ABB RobotStudio station: CakeServer.rspag

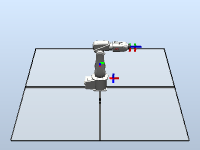
--- station ---
Station Solution2 (saved by RobotStudio 7.0.8460.151)
Controller Vinnie
  mechanical unit ROB_1: IRB120_3_58__01, 6 joints, base frame (0, 0, 0) mm
Layout (positions relative to the parent item):
  - IRB120_3_58__01 [mechanism, from Robots\IRB120_3_58_G_01.rslib] at (0, 0, 0) mm; joint values [0, 0, 0, 0, 0, 0] (rad or m)
Targets, tools, work objects and paths stored in the station and not in the controller backup, written as RAPID:
! task T_ROB1
MODULE MTRN4230_IO_Sample
  PROC MainIO()
    TurnVacOn;
    WaitTime 2;
    TurnVacOff;
    TurnConOnSafely;
    WaitTime 2;
    TurnConOff;
  ENDPROC
  PROC TurnVacOff()
    SetDO DO10_1,0;
  ENDPROC
  PROC TurnConOff()
    SetDO DO10_3,0;
  ENDPROC
  PROC TurnVacOn()
    SetDO DO10_1,1;
  ENDPROC
  PROC TurnConOnSafely()
    SetDO DO10_3,1;
    SetDO DO10_3,0;
  ENDPROC
ENDMODULE


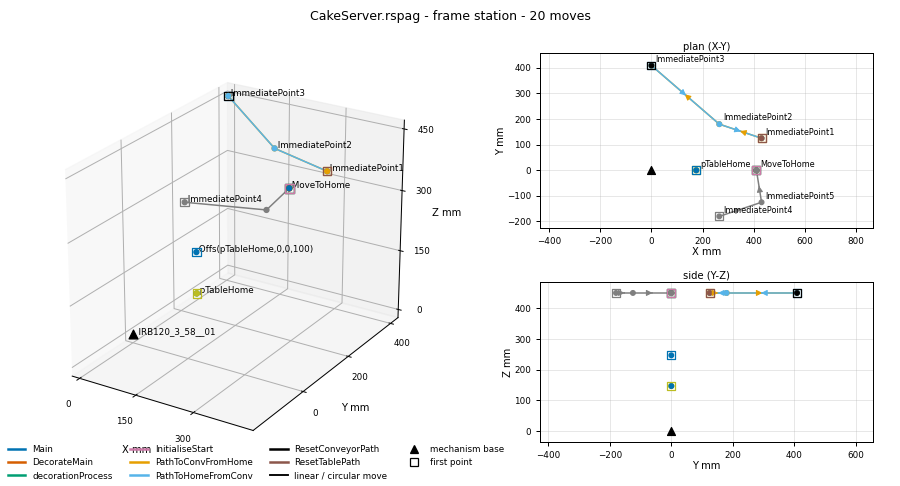
[picture p0: tool path of CakeServer.rspag in frame station, 20 of 38 moves have a stored position in this frame; points joined in program order, loops and branches not executed]
--- Backups/Vinnie/RAPID/TASK1/PROGMOD/CakeShopRobotMain.mod ---
MODULE CakeShopRobotMain
    !***********************************************************
    !
    ! Module: Main robot controller
    ! Author: Rachel Feng, z5112668
    !
    ! Description:
    !   This module is the main controller of all robot movements.
    !   Contains ongoing error checking.
    !   Calls functions to decorate the cake with blocks & icing.
    !   After each pick and place, communicate back to server to see
    !   if decoration is completed.
    !
    !***********************************************************

    ! Interrupts for emergency stops
!    VAR intnum lightCurtain;
!    VAR intnum emergencyStop;
!    VAR intnum emergencyStopMotor;
    VAR num tempConv;
    VAR num response;

    ! Flags to send error message back to GUI
    PERS bool lightCurtainError:=FALSE;
    PERS bool emergencyStopError:=FALSE;
    PERS bool conveyorError:=FALSE;
    PERS bool vacuumError:=FALSE;
    PERS bool clearMessage:=FALSE;

    ! Data received from server
    PERS num letterArrayCopy{3,100,1000};
    PERS num blockArrayCopy{50,7};
    PERS num leftOverArrayCopy{50,6};

    PERS num numLettersCopy;
    PERS num numCoordinatesCopy{100};
    VAR num z_coord:=147.5;

    PERS num numBlocksCopy;
    PERS num numLeftOverCopy;

    ! Flags to check
    PERS bool chocBlocks;
    PERS bool isDecorDone;
    PERS bool letters;
    PERS bool robotMoving;
    PERS bool pauseResume;
    PERS bool stopFlag;

    VAR bool firstConvMove:=FALSE;

    CONST jointtarget removeSingularities := [[0,0,0,0,3,3],[9E+09,9E+09,9E+09,9E+09,9E+09,9E+09]];

    PROC Main()
        ! set up interrups
!        CONNECT timerInt WITH checkTime;
!        ITimer 5,timerInt;
!        ISleep timerInt;

!        CONNECT lightCurtain WITH lTrap;
!        CONNECT emergencyStop WITH eTrap;
!        CONNECT emergencyStopMotor WITH eTrapMotor;

!        ISignalDO\Single,DO_LIGHT_CURTAIN,0,lightCurtain;
!        ISignalDO\Single,DO_ESTOP,1,emergencyStop;
!        ISignalDO\Single,DO_ESTOP2,0,emergencyStopMotor;

        ! Testing stuff
!        ConveyorTestMove01;
!        WaitTime 2;
!        ConveyorTestMove02;
!        WaitTime 2;
!        testVacuumOnOff;
!        WaitTime 2;
!        testSuctionCup;
!        WaitTime 2;
!        DecorTest;
!        WaitTime 2;
!        InkPrintingMain;

        ! stop all functions, return robot arm to home position
        IF stopFlag=TRUE THEN
            turnOffConveyor;
            turnOffGripper;
            turnOffVacuum;
            MoveL MoveToHome,v1000,z100,tool0\WObj:=wobj0;
            StopMove;
            EXIT;
        ENDIF

        ! pause/resume loop
        IF pauseResume=FALSE THEN
            StopMove;
            IF DOutput(DO10_3)=1 THEN
                turnOffConveyor;
                tempConv:=1;
            ENDIF
            WHILE pauseResume=FALSE DO
                ! do nothing
            ENDWHILE
            IF tempConv=1 THEN
                turnOnConveyor;
                tempConv:=0;
            ENDIF
            StartMove;
        ENDIF

        ! move conveyor for first choc block picture
        IF firstConvMove=FALSE THEN
            setDirToRobot;
            turnOnConveyor;
            WaitTime 5;
            turnOffConveyor;
            firstConvMove:=TRUE;
            robotMoving:=FALSE;
        ENDIF

        ! main decoration routine
        IF chocBlocks=TRUE THEN
            DecorateMain blockArrayCopy;
            DecorateMain leftOverArrayCopy;
            chocBlocks:=FALSE;
            turnOnConveyor;
            WaitTime 1;
            turnOffConveyor;
            robotMoving:=FALSE;
        ENDIF

        ! main lettering/icing routine
        IF letters=TRUE THEN
            draw_letter letterArrayCopy, sizes ,167;
            letters:=FALSE;
        ENDIF

        ! delete interrupts (temp)
!        IDelete timerInt;
!        IDelete emergencyStop;
!        IDelete emergencyStopMotor;
!        IDelete lightCurtain;
    ENDPROC

!    ! light curtain trap routine
!    TRAP lTrap
!        ! stop the robot & conveyor
!        StopMove;
!        IF DOutput(DO10_3)=1 THEN
!            turnOffConveyor;
!            tempConv:=1;
!        ENDIF
!        ! print message to gui
!        lightCurtainError:=TRUE;
!        ! print message to flex pendant
!        TPErase;
!        TPWrite "Light curtain obstruction";
!        TPReadFK response,"Please remove obstruction",stEmpty,stEmpty,stEmpty,"No","Fixed";
!        IF response=4 THEN
!            TPErase;
!            TPWrite "Exiting program...";
!            WaitTime 2;
!            EXIT;
!        ELSEIF response=5 THEN
!            TPErase;
!            TPWrite "Resuming...";
!            clearMessage:=TRUE;
!        ENDIF
!        StartMove;
!        IF tempConv=1 THEN
!            turnOnConveyor;
!            tempConv:=0;
!        ENDIF
!        lightCurtainError:=FALSE;
!        RETURN ;
!    ENDTRAP

!    ! emergency stop interrupt for red buttons except motor
!    TRAP eTrap
!        ! stop the robot
!        StopMove;
!        IF DOutput(DO10_3)=1 THEN
!            turnOffConveyor;
!            tempConv:=1;
!        ENDIF
!        ! print message to gui
!        emergencyStopError:=TRUE;
!        ! print message to flex pendant
!        TPErase;
!        TPWrite "Emergency stop!";
!        TPWrite "Please remove any obstructions and hazards from the robot.";
!        TPWrite "Don't forget to reset the light curtain.";
!        TPReadFK response,"Restart?",stEmpty,stEmpty,stEmpty,"No","Yes";
!        IF response=4 THEN
!            TPErase;
!            TPWrite "Exiting program...";
!            WaitTime 2;
!            EXIT;
!        ELSEIF response=5 THEN
!            TPErase;
!            TPWrite "Resuming...";
!            clearMessage:=TRUE;
!        ENDIF
!        StartMove;
!        IF tempConv=1 THEN
!            turnOnConveyor;
!            tempConv:=0;
!        ENDIF
!        emergencyStopError:=FALSE;
!        RETURN ;
!    ENDTRAP

!    ! emergency stop interrupt for motor button
!    TRAP eTrapMotor
!        ! stop the robot
!        StopMove;
!        IF DOutput(DO10_3)=1 THEN
!            turnOffConveyor;
!            tempConv:=1;
!        ENDIF
!        ! print message to gui
!        emergencyStopError:=TRUE;
!        ! print message to flex pendant
!        TPErase;
!        TPWrite "Motor stop!";
!        TPWrite "Please remove any obstructions and hazards from the robot.";
!        TPWrite "Don't forget to reset the light curtain.";
!        TPReadFK response,"Restart?",stEmpty,stEmpty,stEmpty,"No","Yes";
!        IF response=4 THEN
!            TPErase;
!            TPWrite "Exiting program...";
!            WaitTime 2;
!            EXIT;
!        ELSEIF response=5 THEN
!            TPErase;
!            TPWrite "Resuming...";
!            clearMessage:=TRUE;
!        ENDIF
!        StartMove;
!        IF tempConv=1 THEN
!            turnOnConveyor;
!            tempConv:=0;
!        ENDIF
!        emergencyStopError:=FALSE;
!        RETURN ;
!    ENDTRAP

ENDMODULE

--- Backups/Vinnie/RAPID/TASK1/PROGMOD/ConveyorController.mod ---
MODULE ConveyorController
    !***********************************************************
    !
    ! Module: Conveyor Controller
    ! Author: Rachel Feng, z5112668
    !
    ! Description:
    !   This is a module containing all conveyor commands to be called by other modules
    !
    !***********************************************************

    ! Response from error provided from the user
    !VAR num convResp;
    ! Error number for conveyor movement fail
    !VAR errnum CONV_MOVE_ERR:=-1;

    PROC turnOnConveyor()
        !BookErrNo CONV_MOVE_ERR;
        ! if conveyor status (constat) is 1, good to go
        !IF DI10_1=1 THEN
            SetDO DO10_3,1;
        !ELSE
        !    turnOffConveyor;
        !    RAISE CONV_MOVE_ERR;
        !ENDIF

!    ERROR
!        ! Conveyor error: occurs when attempt to turn on conveyor occured when IO/Light Curtain/Cage is not ready/set up
!        IF ERRNO=CONV_MOVE_ERR THEN
!            ! print to gui
!            conveyorError:=TRUE;
!            ! print message to flex pendant
!            TPErase;
!            TPWrite "Please check light curtain and conveyor guard then restart conveyor";
!            TPReadFK convResp,"Checked?",stEmpty,stEmpty,stEmpty,"No","Yes";
!            IF convResp=4 THEN
!                convResp:=0;
!                TPErase;
!                TPWrite "Exiting...";
!                EXIT;
!            ELSEIF convResp=5 THEN
!                convResp:=0;
!                clearMessage:=TRUE;
!                TPErase;
!                TPWrite "Retrying...";
!                conveyorError:=FALSE;
!                RETRY;
!            ENDIF
!        ENDIF
    ENDPROC

    PROC turnOffConveyor()
        SetDO DO10_3,0;
    ENDPROC

    PROC setDirToRobot()
        SetDO DO10_4,1;
    ENDPROC

    PROC setDirFromRobot()
        ! default
        SetDO DO10_4,0;
    ENDPROC
ENDMODULE

--- Backups/Vinnie/RAPID/TASK1/PROGMOD/DecorationPickAndPlace.mod ---
MODULE DecorationPickAndPlace
    !***********************************************************
    !
    ! Module: Decoration Movement Code for Robot
    ! Author: Dylan Dam, z5115759
    !
    ! Description:
    !    This module is responsible for the pick and place for the qwirkle decoration.
    !    The function takes an array that contains the start and end coordinates of the
    !    blocks as well as it's orientation. The robot then moves via a set path that is
    !    defined and proceeds to move to the location of the block on the conveyor belt.
    !    After picking up the block the arm traverses back via the same path and places
    !    the block down. There is a function that rotates axis 6 for blocks that are
    !    orientated differently. After the execution of the place and drop the robot
    !    moves back to the home position.
    !
    ! Inputs:
    !   array - a nx6 or nx7 matrix data, recevied from GUI part, see GUI for more info
    !
    !***********************************************************

    ! Custom waypoints that I have selected
    CONST robtarget ImmediatePoint1:=[[430,125,450],[0,0,1,0],[0,-1,0,0],[9E+09,9E+09,9E+09,9E+09,9E+09,9E+09]];
    CONST robtarget ImmediatePoint2:=[[265,180,450],[0,0,1,0],[0,-1,0,0],[9E+09,9E+09,9E+09,9E+09,9E+09,9E+09]];
    CONST robtarget ImmediatePoint3:=[[0,409,450],[0,0,1,0],[1,-1,1,0],[9E+09,9E+09,9E+09,9E+09,9E+09,9E+09]];
    CONST robtarget ImmediatePoint4:=[[265,-180,450],[0,0,1,0],[1,-1,1,0],[9E+09,9E+09,9E+09,9E+09,9E+09,9E+09]];
    CONST robtarget ImmediatePoint5:=[[430,-125,450],[0,0,1,0],[1,-1,1,0],[9E+09,9E+09,9E+09,9E+09,9E+09,9E+09]];
    CONST robtarget MoveToHome:=[[410,0,450],[0,0,-1,0],[0,0,-1,0],[9E+09,9E+09,9E+09,9E+09,9E+09,9E+09]];
    ! Offset for the end-effector
    CONST num offSet := 75;
    !Dummy Array for Testing
    !CONST num qwirkleArray{4,7} := [[175,0,147,0,409,22.1,45],[548.6,0,147,0,409,22.1,0],[175,520,147,0,409,22.1,-45],[175,-300,147,0,409,22.1,-45]];
    CONST num qwirkleArray{1,7} := [[175,-50,147,0,409,22.1,-89]];

    PROC DecorateMain(num array{*,*})
        TPWRite "Decorating...";
        MoveAbsJ removeSingularities,v400,fine,tool0;
        MoveL MoveToHome,v1000,z100,tool0\WObj:=wobj0;
        WaitTime 1;
        decorationProcess array;
        WaitTime 1;
        MoveL MoveToHome,v1000,z100,tool0\WObj:=wobj0;
        WaitTime 1;
    ENDPROC

    PROC decorationProcess(num array{*,*})

        VAR num xStart;
        VAR num yStart;
        VAR num zStart;
        VAR num xEnd;
        VAR num yEnd;
        VAR num zEnd;
        VAR num orientation;
        VAR robtarget qwirkleLocation;
        VAR robtarget qwirklePlacement;

        FOR a FROM 1 TO Dim(array,1) DO
            ! This part reads in the first line.
            xStart := array{a,4};
            yStart := array{a,5};
            IF xStart = 0 AND yStart = 0 THEN
                ExitCycle;
            ENDIF
            !zStart := array{a,6}+offSet;
            zStart := 22.1+offSet;
            xEnd := array{a,1};
            yEnd := array{a,2};
            zEnd := 147+offSet;
            orientation := array{a,7};

            qwirkleLocation := [[xStart,yStart,zStart],[0,0,1,0],[0,0,0,0],[9E+09,9E+09,9E+09,9E+09,9E+09,9E+09]];
            qwirklePlacement :=[[xEnd,yEnd,zEnd],[0,0,1,0],[0,0,0,0],[9E+09,9E+09,9E+09,9E+09,9E+09,9E+09]];

            PathToConvFromHome;
            MoveL qwirkleLocation,v1000,z100,tool0\WObj:=wobj0;
            WaitTime 1;
            turnOnVacuum;
            turnOnGripper;
            ResetConveyorPath;
            PathToHomeFromConv;
            WaitTime 1;
            MoveL qwirklePlacement,v1000,z100,tool0\WObj:=wobj0;
            RotateTool orientation,qwirklePlacement;
            IF (yEnd < -400) THEN
                LeftSidePath;
            ELSE
                MoveL MoveToHome,v1000,z100,tool0\WObj:=wobj0;
            ENDIF

        ENDFOR

    ENDPROC

    PROC InitialiseStart()
        MoveL MoveToHome,v1000,z100,tool0\WObj:=wobj0;
    ENDPROC

    PROC PathToConvFromHome()
            MoveL ImmediatePoint1,v1000,z100,tool0\WObj:=wobj0;
            MoveL ImmediatePoint2,v1000,z100,tool0\WObj:=wobj0;
            MoveL ImmediatePoint3,v1000,z100,tool0\WObj:=wobj0;
    ENDPROC

    PROC PathToHomeFromConv()
        MoveL ImmediatePoint3,v1000,z100,tool0\WObj:=wobj0;
        MoveL ImmediatePoint2,v1000,z100,tool0\WObj:=wobj0;
        MoveL ImmediatePoint1,v1000,z100,tool0\WObj:=wobj0;
    ENDPROC
    PROC ResetConveyorPath()
        MoveL ImmediatePoint3,v1000,z100,tool0\WObj:=wobj0;
    ENDPROC
    PROC ResetTablePath()
        MoveL ImmediatePoint1,v1000,z100,tool0\WObj:=wobj0;
    ENDPROC

    PROC RotateTool(num Orientation,robtarget a)
        IF Orientation > 90 THEN
            Orientation := 90 - Orientation;
            MoveL RelTool(a,0,0,0,\Rz:= Orientation),v1000,fine,tool0\WObj:=wobj0;
            WaitTime 1;
            turnOffGripper;
            turnOffVacuum;
            WaitTime 1;
        ELSE
            MoveL RelTool(a,0,0,0,\Rz:= Orientation),v1000,fine,tool0\WObj:=wobj0;
            WaitTime 1;
            turnOffGripper;
            turnOffVacuum;
            WaitTime 1;
        ENDIF

    ENDPROC

    PROC LeftSidePath()

        MoveL ImmediatePoint4,v1000,z100,tool0\WObj:=wobj0;
        MoveL ImmediatePoint5,v1000,z100,tool0\WObj:=wobj0;
        MoveL MoveToHome,v1000,z100,tool0\WObj:=wobj0;


    ENDPROC

ENDMODULE

--- Backups/Vinnie/RAPID/TASK1/PROGMOD/InkPrinting.mod ---
MODULE InkPrinting
    !***********************************************************
    !
    ! Module: Ink Printing
    ! Author: Mike Ni, z5083683
    !
    ! Description:
    !   Runs program to move TCP along a given trajectory with a given speed decided by boldness of letter
    !
    ! Input:
    !   data_matrix - a 3xnxm matrix data, recevied from GUI part, see GUI for more info
    !   z_coor - the z coordinate for ink printing, assume to be 147.5
    !
    !***********************************************************

    PERS num x_array{135,1};
    PERS num y_array{135,1};
    PERS num z_array;
    PERS num letterArray{3,8,135};
    PERS num sizes{8};
    ! boldness 0 - unbolded, 1 - bolded
    PERS num bolded{8};
    PERS num boldness;
    ! The Main procedure. When you select 'PP to Main' on the FlexPendant, it will go to this procedure.
    PROC InkPrintingMain()

        ! This is a procedure defined in a System Module, so you will have access to it.
        ! This will move the robot to its calibration.
         MoveToCalibPos;

        ! Call a procedure that we have defined below.
         MoveJSample;

        ! Call another procedure that we have defined.
        ! MoveLSample;
        Path_10;
        !draw_path;
        draw_letter letterArray, sizes, 167;
        !Path_10;

        ! Call another procedure, but provide some input arguments.
        ! VariableSample pTableHome, 100, 100, 0, v100, fine;

        MoveToCalibPos;
    ENDPROC

    PROC draw_path()
        VAR num x;
        VAR num y;
        VAR num z;
        VAR num x_next;
        VAR num y_next;
        VAR pos curr;
        VAR pos next;
        VAR pos prev;
        VAR robtarget pathLoc;
        VAR num distance_from_next;
        VAR num displacement;
        VAR num time_req;
        FOR i FROM 1 TO DIM(x_array,1) DO
            x := x_array{i, 1};
            y := y_array{i, 1};
            ! find next point, except for last point
            IF i <> DIM(x_array, 1) THEN
                x_next := x_array{i+1, 1};
                y_next := y_array{i+1, 1};
            ELSE
                x_next := x;
                y_next := y;
            ENDIF
            z := z_array;
            curr := [x, y, z];
            next := [x_next, y_next, z];
            distance_from_next := Distance(curr, next);
            ! find previous point, start from i = 2
            IF i > 1 THEN
                prev := [x_array{i-1, 1}, x_array{i-1, 1}, z];
                displacement :=  Distance(CPos(\Tool:=tSCup \WObj:=wobj0), curr);
            ENDIF
            pathLoc := [[x, y, z],[0,0,-1,0],[0,0,0,0],[9E9,9E9,9E9,9E9,9E9,9E9]];
            ! check boldness to set speed. 0 - 50mm/s; 1 - 100mm/s
            IF boldness = 0 THEN
                time_req := displacement / 50;
                MoveL pathLoc, v50, z0, tSCup;
                !MoveL pathLoc, v50, \T:=1, fine, tSCup;
            ELSE
                time_req := displacement / 100;
                MoveL pathLoc, v100, z0, tSCup;
                !MoveL pathLoc, v100, \T:= 1, fine, tSCup;
            ENDIF
            !if next point is very far away, move tcp away from object surface
            IF distance_from_next > 15 THEN
                pathLoc := [[x, y, z+50],[0,0,-1,0],[0,0,0,0],[9E9,9E9,9E9,9E9,9E9,9E9]];
                MoveL pathLoc, vmax, \T:=0.1, fine, tSCup;
            ENDIF
        ENDFOR
        !move tcp away once all movement done
        pathLoc := [[x, y, z+10],[0,0,-1,0],[0,0,0,0],[9E9,9E9,9E9,9E9,9E9,9E9]];
        MoveL pathLoc, vmax, \T:=0.1, fine, tSCup;
    ENDPROC

    !use "draw_letter data_matrix" to run
    PROC draw_letter(num data_matrix{*,*,*}, num sizeOfLetter{*}, num z_coor)
        VAR num x;
        VAR num y;
        VAR num z;
        VAR num x_next;
        VAR num y_next;
        VAR pos curr;
        VAR pos next;
        VAR pos prev;
        VAR robtarget pathLoc;
        VAR num distance_from_next;
        VAR num displacement;
        VAR num time_req;
        VAR num bolded;
        VAR speeddata speed;
        MoveAbsJ removeSingularities,v400,fine,tool0;
        FOR index FROM 1 TO DIM(data_matrix,2) DO
            bolded := data_matrix{1,index,1};
            IF bolded = 0 THEN
                speed := [50, 500, 5000, 1000];
            ELSE
                speed := [100, 500, 5000, 1000];
            ENDIF
            FOR i FROM 1 TO sizeOfLetter{index} DO
                x := data_matrix{2,index,i};
                y := data_matrix{3,index,i};

                ! find next point, except for last point
                IF i <> DIM(data_matrix,3) THEN
                    x_next := data_matrix{2,index,i+1};
                    y_next := data_matrix{3,index,i+1};
                ELSE
                    x_next := x;
                    y_next := y;
                ENDIF
                z := z_coor;
                curr := [x, y, z];
                next := [x_next, y_next, z];
                distance_from_next := Distance(curr, next);
                ! find previous point, start from i = 2
                IF i > 1 THEN
                    prev := [data_matrix{2,index,i-1}, data_matrix{3,index,i-1}, z];
                    displacement :=  Distance(CPos(\Tool:=tSCup \WObj:=wobj0), curr);
                ENDIF
                pathLoc := [[x, y, z],[0,0,-1,0],[0,0,0,0],[9E9,9E9,9E9,9E9,9E9,9E9]];
                ! check boldness to set speed. 0 - 50mm/s; 1 - 100mm/s

                MoveL pathLoc, speed, z0, tSCup;

                !if next point is very far away, move tcp away from object surface
                IF distance_from_next > 15 THEN
                    pathLoc := [[x, y, z+50],[0,0,-1,0],[0,0,0,0],[9E9,9E9,9E9,9E9,9E9,9E9]];
                    MoveL pathLoc, vmax, \T:=0.1, fine, tSCup;
                ENDIF
            ENDFOR
            !move tcp away once all movement done
            pathLoc := [[x, y, z+10],[0,0,-1,0],[0,0,0,0],[9E9,9E9,9E9,9E9,9E9,9E9]];
            MoveL pathLoc, vmax, \T:=0.1, fine, tSCup;
        ENDFOR
    ENDPROC

    PROC Path_10()
        !Defines the trajectory coordinates
        VAR num step_count := 0;
        bolded := [0,1,0,1,0,1,0,1];
        boldness := 0;
        x_array := [
        [347.3852228],
        [340.1824253],
        [332.9796278],
        [325.7768303],
        [319.2288325],
        [312.026035],
        [304.8232375],
        [309.4068359],
        [315.9548336],
        [322.5028314],
        [329.0508291],
        [335.5988269],
        [342.1468246],
        [300.2396391],
        [306.7876368],
        [313.9904343],
        [321.1932318],
        [327.7412296],
        [334.9440271],
        [341.4920249],
        [302.8588381],
        [308.7520361],
        [315.3000339],
        [321.8480316],
        [328.3960294],
        [334.9440271],
        [341.4920249],
        [304.1684377],
        [304.8232375],
        [304.8232375],
        [304.8232375],
        [350.0044219],
        [344.111224],
        [336.9084264],
        [329.7056289],
        [322.5028314],
        [315.3000339],
        [308.0972363],
        [348.0400226],
        [340.8372251],
        [333.6344276],
        [326.43163],
        [325.1220305],
        [325.7768303],
        [331.0152285],
        [337.5632262],
        [344.7660237],
        [324.4672307],
        [319.2288325],
        [312.6808348],
        [306.132837],
        [302.8588381],
        [302.2040384],
        [305.4780372],
        [312.6808348],
        [319.8836323],
        [302.2040384],
        [307.4424366],
        [312.6808348],
        [319.2288325],
        [325.7768303],
        [332.324828],
        [338.8728258],
        [344.7660237],
        [304.8232375],
        [311.3712352],
        [318.5740327],
        [325.7768303],
        [332.324828],
        [338.8728258],
        [350.0044219],
        [343.4564242],
        [336.2536267],
        [329.0508291],
        [321.8480316],
        [314.6452341],
        [350.0044219],
        [336.9084264],
        [341.4920249],
        [348.6948224],
        [304.1684377],
        [310.7164354],
        [317.919233],
        [325.1220305],
        [332.324828],
        [336.2536267],
        [336.2536267],
        [329.7056289],
        [323.1576312],
        [316.6096334],
        [310.7164354],
        [304.8232375],
        [351.3140215],
        [346.0756233],
        [348.6948224],
        [348.6948224],
        [312.6808348],
        [307.4424366],
        [306.132837],
        [310.7164354],
        [317.2644332],
        [323.8124309],
        [329.0508291],
        [334.2892273],
        [340.1824253],
        [343.4564242],
        [349.3496222],
        [351.3140215],
        [348.6948224],
        [342.8016244],
        [335.5988269],
        [329.0508291],
        [322.5028314],
        [315.9548336],
        [309.4068359],
        [304.8232375],
        [305.4780372],
        [310.7164354],
        [325.7768303],
        [321.8480316],
        [315.3000339],
        [308.7520361],
        [306.7876368],
        [310.0616357],
        [316.6096334],
        [323.1576312],
        [330.3604287],
        [336.9084264],
        [343.4564242],
        [348.6948224],
        [349.3496222],
        [344.7660237],
        [338.218026],
        [331.6700282],
        [324.4672307]
        ];

        y_array := [
        [137.4530852],
        [137.4530852],
        [137.4530852],
        [137.4530852],
        [136.800876],
        [136.800876],
        [136.800876],
        [131.5832025],
        [130.2787841],
        [128.9743658],
        [127.6699474],
        [126.3655291],
        [125.0611107],
        [104.842626],
        [106.7992536],
        [106.7992536],
        [106.7992536],
        [106.7992536],
        [106.7992536],
        [107.4514628],
        [108.103672],
        [111.3647179],
        [113.3213454],
        [115.277973],
        [117.2346005],
        [118.5390189],
        [119.8434372],
        [94.40727912],
        [87.23297812],
        [80.05867712],
        [72.88437611],
        [80.7108863],
        [83.97193221],
        [83.97193221],
        [83.97193221],
        [83.97193221],
        [83.97193221],
        [83.97193221],
        [61.14461083],
        [61.14461083],
        [61.14461083],
        [60.49240165],
        [53.97030983],
        [46.79600882],
        [42.23054455],
        [41.57833537],
        [41.57833537],
        [46.79600882],
        [41.57833537],
        [40.92612618],
        [42.88275373],
        [48.75263637],
        [55.27472819],
        [61.14461083],
        [61.14461083],
        [61.14461083],
        [29.1863609],
        [24.62089663],
        [20.05543235],
        [17.44659562],
        [15.48996808],
        [12.88113135],
        [9.620085438],
        [6.359039527],
        [3.750202798],
        [4.40241198],
        [4.40241198],
        [4.40241198],
        [3.750202798],
        [5.706830344],
        [24.62089663],
        [27.22973336],
        [27.22973336],
        [27.22973336],
        [27.22973336],
        [26.57752417],
        [-25.5992104],
        [-30.81688386],
        [-25.5992104],
        [-25.5992104],
        [-26.25141958],
        [-25.5992104],
        [-25.5992104],
        [-25.5992104],
        [-25.5992104],
        [-19.72932776],
        [-12.55502676],
        [-10.59839921],
        [-13.85944512],
        [-17.12049103],
        [-20.38153694],
        [-24.29479204],
        [-36.6867665],
        [-41.90443996],
        [-48.42653178],
        [-55.60083278],
        [-40.60002159],
        [-45.16548587],
        [-51.68757769],
        [-57.55746033],
        [-58.20966951],
        [-56.25304197],
        [-51.68757769],
        [-47.12211341],
        [-43.20885832],
        [-68.64501643],
        [-71.90606234],
        [-78.42815416],
        [-84.95024598],
        [-88.21129189],
        [-88.21129189],
        [-85.60245516],
        [-84.95024598],
        [-87.55908271],
        [-86.90687353],
        [-81.68920007],
        [-74.51489907],
        [-69.94943479],
        [-77.1237358],
        [-100.6032664],
        [-101.9076847],
        [-105.1687306],
        [-111.6908225],
        [-118.2129143],
        [-120.1695418],
        [-120.821751],
        [-120.821751],
        [-120.1695418],
        [-118.8651235],
        [-114.2996592],
        [-107.7775674],
        [-102.5598939],
        [-101.2554755],
        [-100.6032664],
        [-100.6032664]
        ];

        sizes:=[27,11,18,20,16,13,14,16];
        z_array := 147;
        FOR i FROM 1 TO 27 DO
            letterArray{1,1,1} := bolded{1};
            letterArray{2,1,i} := x_array{i+step_count,1};
            letterArray{3,1,i} := y_array{i+step_count,1};
        ENDFOR
        step_count := 27;
        FOR i FROM 1 TO 11 DO
            letterArray{1,2,1} := bolded{2};
            letterArray{2,2,i} := x_array{i+step_count,1};
            letterArray{3,2,i} := y_array{i+step_count,1};
        ENDFOR
        step_count := 38;
        FOR i FROM 1 TO 18 DO
            letterArray{1,3,1} := bolded{3};
            letterArray{2,3,i} := x_array{i+step_count,1};
            letterArray{3,3,i} := y_array{i+step_count,1};
        ENDFOR
        step_count := 56;
        FOR i FROM 1 TO 20 DO
            letterArray{1,4,1} := bolded{4};
            letterArray{2,4,i} := x_array{i+step_count,1};
            letterArray{3,4,i} := y_array{i+step_count,1};
        ENDFOR
        step_count := 76;
        FOR i FROM 1 TO 16 DO
            letterArray{1,5,1} := bolded{5};
            letterArray{2,5,i} := x_array{i+step_count,1};
            letterArray{3,6,i} := y_array{i+step_count,1};
        ENDFOR
        step_count := 92;
        FOR i FROM 1 TO 13 DO
            letterArray{1,6,1} := bolded{6};
            letterArray{2,6,i} := x_array{i+step_count,1};
            letterArray{3,6,i} := y_array{i+step_count,1};
        ENDFOR
        step_count := 105;
        FOR i FROM 1 TO 14 DO
            letterArray{1,7,1} := bolded{7};
            letterArray{2,7,i} := x_array{i+step_count,1};
            letterArray{3,7,i} := y_array{i+step_count,1};
        ENDFOR
        step_count := 119;
        FOR i FROM 1 TO 16 DO
            letterArray{1,8,1} := bolded{8};
            letterArray{2,8,i} := x_array{i+step_count,1};
            letterArray{3,8,i} := y_array{i+step_count,1};
        ENDFOR
        !FOR i FROM 1 TO DIM(x_array, 1) DO
        !    letterArray{2,1,i} := x_array{i,1};
        !    letterArray{3,1,i} := y_array{i,1};
        !ENDFOR
    ENDPROC

    PROC MoveJSample()

        ! 'MoveJ' executes a joint motion towards a robtarget. This is used to move the robot quickly from one point to another when that
        !   movement does not need to be in a straight line.
        ! 'pTableHome' is a robtarget defined in system module. The exact location of this on the table has been provided to you.
        ! 'v100' is a speeddata variable, and defines how fast the robot should move. The numbers is the speed in mm/sec, in this case 100mm/sec.
        ! 'fine' is a zonedata variable, and defines how close the robot should move to a point before executing its next command.
        !   'fine' means very close, other values such as 'z10' or 'z50', will move within 10mm and 50mm respectively before executing the next command.
        ! 'tSCup' is a tooldata variable. This has been defined in a system module, and represents the tip of the suction cup, telling the robot that we
        !   want to move this point to the specified robtarget. Please be careful about what tool you use, as using the incorrect tool will result in
        !   the robot not moving where you would expect it to. Generally you should be using
        MoveJ pTableHome, v100, \T:=0.5, fine, tSCup;

    ENDPROC

    PROC MoveLSample()

        ! 'MoveL' will move in a straight line between 2 points. This should be used as you approach to pick up a chocolate
        ! 'Offs' is a function that is used to offset an existing robtarget by a specified x, y, and z. Here it will be offset 100mm in the positive z direction.
        !   Note that function are called using brackets, whilst procedures and called without brackets.
        MoveL Offs(pTableHome, 0, 0, 100), v100, fine, tSCup;

    ENDPROC

    PROC VariableSample(robtarget target, num x_offset, num y_offset, num z_offset, speeddata speed, zonedata zone)

        ! Call 'MoveL' with the input arguments provided.
        MoveL Offs(target, x_offset, y_offset, z_offset), speed, zone, tSCup;

    ENDPROC

ENDMODULE

--- Backups/Vinnie/RAPID/TASK1/PROGMOD/VacuumController.mod ---
MODULE VacuumController
    !***********************************************************
    !
    ! Module: Vacuum Controller
    ! Author: Rachel Feng, z5112668
    !
    ! Description:
    !   This is a module containing all vacuum commands to be called by other modules
    !
    !***********************************************************

    ! Response from error provided by the user
    VAR num vacResp;
    ! Error number for suction cup fail
    VAR errnum SUCTION_CUP_ERR:=-1;
    ! Timer interrupt
!    VAR intnum timerInt;

    PROC turnOnVacuum()
        SetDO DO10_1,1;
        !        IWatch timerInt;
    ENDPROC

    PROC turnOffVacuum()
!        ISleep timerInt;
        turnOffGripper;
        SetDO DO10_1,0;
    ENDPROC

    PROC turnOnGripper()
        BookErrNo SUCTION_CUP_ERR;
        IF DOutput(DO10_1)=1 THEN
            SetDO DO10_2,1;
        ELSE
            RAISE SUCTION_CUP_ERR;
        ENDIF

    ERROR
        ! Suction cup error: occurs when attempt to activate suction cup occured before vacuum pump activation
        IF ERRNO=SUCTION_CUP_ERR THEN
            ! print message to gui
            vacuumError:=TRUE;
            ! print message to flex pendant
            TPErase;
            TPReadFK vacResp,"Do you want to turn on vacuum?",stEmpty,stEmpty,stEmpty,"No","Yes";
            IF vacResp=4 THEN
                vacResp:=0;
                TPErase;
                TPWrite "Exiting...";
                EXIT;
            ELSEIF vacResp=5 THEN
                vacResp:=0;
                clearMessage:=TRUE;
                TPErase;
                TPWrite "Turning on vacuum";
                turnOnVacuum;
                vacuumError:=FALSE;
                RETRY;
            ENDIF
        ENDIF


    ENDPROC

    PROC turnOffGripper()
        SetDO DO10_2,0;
    ENDPROC

!    TRAP checkTime
!        TPErase;
!        TPWrite "Vacuum was on for too long...";
!        TPWrite "Turning off...";
!        turnOffVacuum;
!        RETURN ;
!    ENDTRAP
ENDMODULE

--- Backups/Vinnie/RAPID/TASK1/SYSMOD/MTRN_Rob_Data.sys ---
MODULE MTRN_Rob_Data (SYSMODULE, NOSTEPIN, READONLY)

 ! PREDEFINED DATA AND ROBOT CELL INFORMATION
 !*******************************************

 ! For the ABB IRB120 Robot in the Mechatronics Blockhouse Lab for the MTRN4230 Robotics Course 2014

 ! TARGETS
 !********

 ! Calibrate Position for all Joints
 CONST jointtarget jtCalibPos:=[[0,0,0,0,0,0],[9E+09,9E+09,9E+09,9E+09,9E+09,9E+09]];

  ! Home Position
 CONST jointtarget jtHomePos:=[[-90,0,0,0,0,0],[9E+09,9E+09,9E+09,9E+09,9E+09,9E+09]];

 ! Home Position of the Table (T1) with tSCup touching Table
 CONST robtarget pTableHome:=[[175,0,147],[0,0,-1,0],[0,0,0,0],[9E+09,9E+09,9E+09,9E+09,9E+09,9E+09]];

 ! Home Position of the Conveyor (C1) with tSCup touching Conveyor
 CONST robtarget pConvHome:=[[0,409,22],[0,-0.7071068,0.7071068,0],[0,0,0,0],[9E+09,9E+09,9E+09,9E+09,9E+09,9E+09]];

 ! Table & Conveyor Dimensions, References & Extent limits as Follows (X,Y,Z in mm):
 !
 !                                                       Conveyor Frame
 !       ------>Y                                   |<-------- 616 -------->|
 !       |                                          |   | Conveyor Belt |   |
 !       |                                          |   |<---- 450 ---->|   |
 !       |                            ||    --------|   |               |   |
 !       v                            \/    |------||   |   0,409,22    |   |
 !       X             Robot Centre  ---->  ||  + |||   |      +        |   |
 !                                          ||    |||   |      C1       |   |
 !     Robot Centre to edge of Table=129    -|    |_|   |               |   |
 !   ----------------------------------------|    |-----------------------------------
 !   |                                /\      ----                                   |
 !   |                                ||      |  |                                   |
 !   |     175,-520,147                     175,0,147                  175,520,147   |
 !   |           +                              +                           +        |
 !   |           T2                             T1                          T3       |
 !   |                                                                               |
 !   |                                                                               |
 !   |                                    548.6,0,147                                |
 !   |                                          +                                    |
 !   |                                          T4                                   |
 !   |                                                                               |
 !   ---------------------------------------------------------------------------------

 ! TOOL DATA
 !**********

 ! Suction Cup Tool Data
 PERS tooldata tSCup:=[TRUE,[[0,0,65],[1,0,0,0]],[0.5,[0,0,20],[1,0,0,0],0,0,0]];
 !
 ! Suction Cup Face is 65mm in Z direction from Tool0

 ! LOAD DATA
 !**********

 ! Chocolate Bar Load Data
 PERS loaddata loChoc:=[0.035,[0,0,3],[1,0,0,0],0,0,0];

 !
 ! Chocolate Bar Weight    : 35g
 !
 ! Chocolate Bar Dimensions: 114.5 x 53 x 7.5mm (Including Perspex substitute in wrapper)
 !
 ! Chocolate Box Dimensions: 214.0 x 119.0 x 46.0mm (Internal)
 !                           219.5 x 121.0 x 48.0mm (External)
 !
 ! Chocolate Box References:
 !
 !                         -------------------------
 !                         |----- ----- ----- -----|
 !                         ||   | |   | |   | |   ||
 !                         ||   | |   | |   | |   ||
 !                         ||B4 | |B3 |+|B2 | |B1 ||
 !                         ||   | |   | |   | |   ||
 !                         ||   | |   | |   | |   ||
 !                         |----- ----- ----- -----|
 !                         -------------------------
 !
 ! NOTE: + marks centre of box and Conveyor Home Position C1

 ! WORK OBJECT DATA
 !*****************
 !                                    [Uframe User co-ord System] [Oframe Object Co-ord System]
 PERS wobjdata wTable:=[FALSE,TRUE,"",[[175,0,147],[1,0,0,0]],[[0,0,0],[1,0,0,0]]];
 PERS wobjdata wConv:=[FALSE,TRUE,"",[[50,184,22],[0.5,-0.5,0.5,0.5]],[[1,1,1],[1,0,0,0]]];

 ! WorkObject orientations for the Table and Conveyor
 !
 !                    |   |               |   |
 !                    |   Y               |   |
 !                    |   ^               |   |
 !             -------|   |               |   |
 !             |     ||   | \Wobj:=vConv  |   |
 !             |  +  ||   |               |   |
 !             |     ||   |               |   |
 !             -------|  Zo------>X       |   |
 !   ---------------------------------------------------
 !               Zo----->Y                             |
 !                |                                    |
 !                | \Wobj:=vTable                      |
 !                |                                    |
 !                v                                    |
 !                X                                    |
 !                                                     |

 ! COMMENTS
 !*********

 ! Digital I/O Names and Functions
 ! DI10-1	ConStat	= Conveyor Status (Active = 1, Inactive = 0)
 !
 ! DO10-1	VacPwr	= Vacuum Power (Run = 1, Stop =0)
 ! DO10-2	VacSol	= Vacuum Solenoid (Open = 1, Closed =0)
 ! D010-3	ConRun	= Conveyer Start (Run = 1, Stop = 0)
 ! D010-4	ConDir	= Conveyer Direction (Towards Robot = 1, Away from Robot = 0)

ENDMODULE

--- Backups/Vinnie/RAPID/TASK1/SYSMOD/MTRN_Rob_Proc.sys ---
MODULE MTRN_Rob_Proc (SYSMODULE, NOSTEPIN, READONLY)

 ! MTRN ROBOTICS COMMON PROCEDURES
 !********************************
 !
 ! For the ABB IRB120 Robot in the Mechatronics Blockhouse Lab for the MTRN4230 Robotics Course 2014
 !

 PROC MoveToCalibPos()
 !***************************************************************************************
 !
 ! Move to Calibrate Position
 !
 !***************************************************************************************

 MoveAbsJ jtCalibPos,v400,fine,tool0;

 ENDPROC

  PROC MoveToHomePos()
 !***************************************************************************************
 !
 ! Move to Calibrate Position
 !
 !***************************************************************************************

 MoveAbsJ jtHomePos,v400,fine,tool0;

 ENDPROC

ENDMODULE

--- Backups/Vinnie/RAPID/TASK2/PROGMOD/CakeShopServer.mod ---
MODULE CakeShopServer
    !***********************************************************
    !
    ! Module: Cake Shop Server
    ! Author: Lawrence Wang, z5075019
    !
    ! Description:
    !    Main server to receive information from Matlab image processing.
    !    Translates received data into arrays for T_ROB
    !
    ! Inputs & Outputs:
    !    See below functions
    !
    !***********************************************************

    ! Tcp socket object
    VAR socketdev client_socket;

    ! The host and port that we will be listening for a connection on. Currently set to localhost.
    PERS string host:="127.0.0.1";
    CONST num port:=1025;

    ! Array of letter coordinates
    ! Dimension 1 is the type of data i.e. 1 = boldness, 2 = x coordinate, 3 = y coordinate
    ! Dimension 2 is the letter number i.e. 1 is the first letter, 5 is the fifth letter
    ! Dimension 3 is the coordinate number in a letter i.e. 3 is the third coordinate
    ! e.g. letterArray{2, 3, 6} refers to the x coordinate of the 6th point in the 3rd letter
    ! e.g. letterArray{1, 6, 1} refers to the boldness of the 6th letter (Dimension 3 is always 1 for boldness)
    VAR num letterArray{3,100,1000};

    ! Array of strings storing the message. Each element is one part (part is a section separated by a comma delimiter)
    VAR string messageArray{10000};
    ! Array of blocks on the cake/conveyor + orientation. Limit of 50 blocks but array may not be filled.
    VAR num blockArray{50,7};
    ! Array of left over blocks on conveyor + junk area.
    VAR num leftOverArray{50,6};
    ! Flag to check if error has occurred. (Not used at the moment)
    VAR bool errorFlag;
    ! String containing error message that needs to be sent
    VAR string errorMessage;

    ! Number of letters in a letterArray. Needed as array size may change and leftover data may still be there.
    VAR num numLetters;
    ! Number of coordinates in path for each letter.
    VAR num numCoordinates{100};

    ! Number of blocks on cake/conveyor. Needed as array size may change.
    VAR num numBlocks;
    ! Number of left over blocks on conveyor.
    VAR num numLeftOver;

    ! Flag to see if a message was received
    VAR bool messageFlag;

    ! A copy of relevant variables above to be shared with T_ROB
    PERS num letterArrayCopy{3,100,1000};
    PERS num blockArrayCopy{50,7};
    PERS num leftOverArrayCopy{50,6};

    PERS num numLettersCopy;
    PERS num numCoordinatesCopy{100};

    PERS num numBlocksCopy;
    PERS num numLeftOverCopy;

    ! Flags so the robot knows which operation to run
    PERS bool chocBlocks:=FALSE;
    PERS bool isDecorDone:=FALSE;
    PERS bool letters:=FALSE;

    ! Flag to determine if more information will be received
    PERS bool robotMoving:=TRUE;

    ! Flag to pause and resume robot operations, TRUE will indicate operations are resumed, FALSE will pause the robot
    PERS bool pauseResume:= TRUE;

    ! Flag to stop  the robot completely, TRUE will stop the robot
    PERS bool stopFlag:= FALSE;

    ! Flags to send error message back to GUI
    PERS bool lightCurtainError;
    PERS bool emergencyStopError;
    PERS bool conveyorError;
    PERS bool vacuumError;
    PERS bool clearMessage;

    VAR intnum lightCurtain;
    VAR intnum emergencyStop;
    VAR intnum emergencyStopMotor;

    VAR num tempConv;
    VAR num response;

    PROC Main()
	IF RobOS()  THEN
	        host:="192.168.125.1";
	ELSE
		host:="127.0.0.1";
	ENDIF
        ListenForAndAcceptConnection client_socket,host,port;
        CONNECT lightCurtain WITH lTrap;
        CONNECT emergencyStop WITH eTrap;
        CONNECT emergencyStopMotor WITH eTrapMotor;

        ISignalDO\Single,DO_LIGHT_CURTAIN,0,lightCurtain;
        ISignalDO\Single,DO_ESTOP,1,emergencyStop;
        ISignalDO\Single,DO_ESTOP2,0,emergencyStopMotor;
        WHILE stopFlag = FALSE DO
            MainServer;
        ENDWHILE
        IDelete emergencyStop;
        IDelete emergencyStopMotor;
        IDelete lightCurtain;
        CloseConnection client_socket;
    ENDPROC

    ! Example of how the functions might be called. Normally start with ListenForAndAcceptConnection to open the socket,
    ! Do all the receiveMessage and sendError.
    ! When the program has finished then call CloseConnection to close the connection.
    PROC MainServer()
        !errorMessage:="errorerror";

        !ListenForAndAcceptConnection client_socket,host,port;
        messageFlag := FALSE;

        receiveMessage client_socket,messageArray;

        IF messageFlag = TRUE THEN
            parseString messageArray,blockArray,leftOverArray,numBlocks,numLeftOver,letterArray,numLetters,numCoordinates;
        ENDIF

        !sendError client_socket,errorMessage;

        IF robotMoving=FALSE THEN
            sendRobotUpdate client_socket,"Take another picture";
        ENDIF

        IF lightCurtainError=TRUE THEN
            sendError client_socket,"Light Curtain Obstruction. Please check Flex Pendant";
        ENDIF
        IF emergencyStopError=TRUE THEN
            sendError client_socket,"Emergency Stop occured. Please check Flex Pendant";
        ENDIF
        IF conveyorError=TRUE THEN
            sendError client_socket,"Conveyor Error. Please check Flex Pendant";
        ENDIF
        IF vacuumError=TRUE THEN
            sendError client_socket,"Vacuum Error. Please check Flex Pendant";
        ENDIF
        IF clearMessage=TRUE THEN
            sendError client_socket,"";
        ENDIF


        ! Send the string back to the client, adding a line feed character.
        ! SocketSend client_socket \Str:=(received_str + "\0A");

        !CloseConnection client_socket;
    ENDPROC

    ! INPUT
    !   socketdev client_socket - this is a socket to be opened and connected to
    !   string host - ip address to connect to e.g. "192.168.0.2" or "127.0.0.1"
    !   num port - port number to connect to e.g. 20000
    ! OUTPUT
    !   socketdev client_socket - the socket has now connected to a client
    PROC ListenForAndAcceptConnection(VAR socketdev client_socket,string host,num port)
        ! Create the socket to listen for a connection on.
        VAR socketdev welcome_socket;
        SocketCreate welcome_socket;

        ! Bind the socket to the host and port.
        SocketBind welcome_socket,host,port;

        ! Listen on the welcome socket.
        SocketListen welcome_socket;

        ! Accept a connection on the host and port.
        SocketAccept welcome_socket,client_socket\Time:=WAIT_MAX;

        ! Close the welcome socket, as it is no longer needed.
        SocketClose welcome_socket;
    ENDPROC

    ! INPUT
    !   socketdev client_socket - socket to be closed
    ! OUTPUT
    !   socketdev client_socket - closed socket
    PROC CloseConnection(VAR socketdev client_socket)
        SocketClose client_socket;
    ENDPROC

    ! INPUT
    !   socketdev client_socket - socket to be read from
    ! OUTPUT
    !   string messageArray{*} - Array of strings which stores all the parts of the message
    PROC receiveMessage(VAR socketdev client_socket,VAR string messageArray{*})
        VAR string received_str;
        VAR num count:=1;
        VAR string end_str:="end";
        VAR string ack_str:="ACK";

        !errorMessage := "errorerror";

        ! Receive a string from the client.
        SocketReceive client_socket\Str:=received_str\Time:=1;
        messageFlag := TRUE;
        messageArray{count}:=received_str;
        SocketSend client_socket\Str:=(ack_str+"\0A");
        count:=count+1;
        WHILE (received_str<>(end_str+"\0A")) DO
            SocketReceive client_socket\Str:=received_str\Time:=WAIT_MAX;
            messageArray{count}:=received_str;
            SocketSend client_socket\Str:=(ack_str+"\0A");
            !            !IF count MOD 2 = 1 THEN
            !               SocketSend client_socket \Str:=(ack_str+"\0A");
            !            ELSE
            !                sendError errorMessage;
            !            ENDIF
            count:=count+1;
        ENDWHILE

        ERROR
            IF ERRNO=ERR_SOCK_CLOSED THEN
                ListenForAndAcceptConnection client_socket,host,port;
                RETRY;
            ENDIF
            IF ERRNO=ERR_SOCK_TIMEOUT THEN
                RETURN;
            ENDIF
    ENDPROC

    ! INPUT
    !   socketdev client_socket - Socket which the message will be sent to.
    !   string errorMessage - error message that will be sent.
    PROC sendError(VAR socketdev client_socket,string errorMessage)
        SocketSend client_socket\Str:=("0, "+errorMessage+"\0A");
    ENDPROC

    ! INPUT
    !   socketdev client_socket - Socket which the message will be sent to.
    !   string message - robot update message that will be sent.
    PROC sendRobotUpdate(VAR socketdev client_socket,string message)
        SocketSend client_socket\Str:=("3, "+message+"\0A");
    ENDPROC

    ! INPUT
    !   string messageArray{*} - Array of strings which contains the message
    ! OUTPUT
    !   num blockArray{*,*} - Array of blocks on the cake/conveyor. Only used when messagetype is for block trajectories
    !   num leftOverArray{*,*} - Array of left over blocks on conveyor and junk area. Only used when messagetype is for block trajectories
    !   num numBlocks - Number of blocks on cake/conveyor. Only used when messagetype is for block trajectories
    !   num numLeftOver - Number of left over blocks. Only used when messagetype is for block trajectories
    !   num letterArray{*,*,*} - Array which contains boldness and letters/numbers. Only used when messagetype is for letter trajectories
    !   num numLetters - Number of letters. Only used when messagetype is for letter trajectories
    !   num numCoordinates{100} - Number of coordinates for each letter. Only used when messagetype is for letter trajectories
    ! NOTES
    !   messagetype is determined by first element of messageArray.
    PROC parseString(VAR string messageArray{*},VAR num blockArray{*,*},VAR num leftOverArray{*,*},VAR num numBlocks,VAR num numLeftOver,VAR num letterArray{*,*,*},VAR num numLetters,VAR num numCoordinates{*})
        IF messageArray{1}="0\0A" THEN

        ELSEIF messageArray{1}="1\0A" THEN
            str2BlockTraj messageArray,blockArray,leftOverArray,numBlocks,numLeftOver;
            blockArrayCopy:=blockArray;
            leftOverArrayCopy:=leftOverArray;
            numBlocksCopy:=numBlocks;
            numLeftOverCopy:=numLeftOver;
            chocBlocks:=TRUE;
            robotMoving:=TRUE;
        ELSEIF messageArray{1}="2\0A" THEN
            str2LetterTraj messageArray,letterArray,numLetters,numCoordinates;
            letterArrayCopy:=letterArray;
            numLettersCopy:=numLetters;
            numCoordinatesCopy:=numCoordinates;
            letters:=TRUE;
        ELSEIF messageArray{1}="4\0A" THEN
            IF pauseResume = TRUE THEN
                pauseResume := FALSE;
            ELSE
                pauseResume := TRUE;
            ENDIF
        ELSEIF messageArray{1} = "5\0A" THEN
            stopFlag := TRUE;

        ENDIF
    ENDPROC

    ! INPUT
    !   string messageArray - Array of strings which contains the message
    ! OUTPUT
    !   num letterArray{*,*,*} - Array which contains boldness and letters/numbers.
    !   num numLetters - Number of letters.
    !   num numCoordinates{100} - Number of coordinates for each letter.
    ! NOTES
    !   This function does not need to be called. Normally done by parseString.
    PROC str2LetterTraj(string messageArray{*},VAR num letterArray{*,*,*},VAR num numLetters,VAR num numCoordinates{*})
        !VAR num numLetters;
        !VAR num numCoordinates{100};
        VAR bool convertStatus;
        !VAR num count;
        !VAR num count2;
        VAR num posInStr;
        VAR num i;
        VAR num j;

        posInStr:=2;
        !number of letters
        convertStatus:=StrToVal(messageArray{posInStr},numLetters);
        posInStr:=posInStr+1;

        !posInStr := 1 + 2
        FOR i FROM 1 TO numLetters DO
            !number of cooridnates for each letter
            convertStatus:=StrToVal(messageArray{posInStr},numCoordinates{i});
            posInStr:=posInStr+1;

        ENDFOR
        !posInStr := 1 + 2 + numLetters
        FOR i FROM 1 TO numLetters DO
            !boldness of letters
            convertStatus:=StrToVal(messageArray{posInStr},letterArray{1,i,1});
            posInStr:=posInStr+1;

        ENDFOR

        !posInStr := 1 + 2 + 2*numLetters;
        FOR i FROM 1 TO numLetters DO
            FOR j FROM 1 TO numCoordinates{i} DO
                ! x coordinate of letters
                convertStatus:=StrToVal(messageArray{posInStr},letterArray{2,i,j});
                posInStr:=posInStr+1;
                ! y coordinate of letters
                convertStatus:=StrToVal(messageArray{posInStr},letterArray{3,i,j});
                posInStr:=posInStr+1;
            ENDFOR

        ENDFOR
    ENDPROC

    ! INPUT
    !   socketdev client_socket - Socket which the message will be sent to.
    ! OUTPUT
    !   num blockArray{*,*} - Array of blocks on the cake/conveyor.
    !   num leftOverArray{*,*} - Array of left over blocks on conveyor and junk area.
    !   num numBlocks - Number of blocks on cake/conveyor.
    !   num numLeftOver - Number of left over blocks.
    ! NOTES
    !   This function does not need to be called. Normally done by parseString.
    PROC str2BlockTraj(string messageArray{*},VAR num blockArray{*,*},VAR num leftOverArray{*,*},VAR num numBlocks,VAR num numLeftOver)
        !VAR num numBlocks;
        !VAR num numLeftOver;
        VAR bool convertStatus;
        !VAR num count;
        VAR num posInStr;
        VAR num i;
        VAR num j;

        posInStr:=2;
        convertStatus:=StrToVal(messageArray{posInStr},numBlocks);
        posInStr:=posInStr+1;
        convertStatus:=StrToVal(messageArray{posInStr},numLeftOver);
        posInStr:=posInStr+1;

        !count := 1;
        FOR i FROM 1 TO numBlocks DO
            FOR j FROM 1 TO 7 DO
                convertStatus:=StrToVal(messageArray{posInStr},blockArray{i,j});
                posInStr:=posInStr+1;
            ENDFOR

            !            ! x coordinate of cake block
            !            convertStatus := StrToVal(messageArray{posInStr},blockArray{i,1});
            !            posInStr := posInStr + 1;
            !            ! y coordinate of cake block
            !            convertStatus := StrToVal(messageArray{posInStr},blockArray{i,2});
            !            posInStr := posInStr + 1;
            !            ! z coordinate of cake block
            !            convertStatus := StrToVal(messageArray{posInStr},blockArray{count,3});
            !            posInStr := posInStr + 1;
            !            ! x coordinate of conveyor block
            !            convertStatus := StrToVal(messageArray{posInStr},blockArray{count,4});
            !            posInStr := posInStr + 1;
            !            ! y coordinate of conveyor block
            !            convertStatus := StrToVal(messageArray{posInStr},blockArray{count,5});
            !            posInStr := posInStr + 1;
            !            ! z coordinate of conveyor block
            !            convertStatus := StrToVal(messageArray{posInStr},blockArray{count,6});
            !            posInStr := posInStr + 1;
            !            ! orientation of block
            !            convertStatus := StrToVal(messageArray{posInStr},blockArray{count,7});
            !            posInStr := posInStr + 1;
            !            count := count + 1;
        ENDFOR

        !count := 1;
        FOR i FROM 1 TO numLeftOver DO
            FOR j FROM 1 TO 6 DO
                convertStatus:=StrToVal(messageArray{posInStr},leftOverArray{i,j});
                posInStr:=posInStr+1;
            ENDFOR
            !            !x coordinate of leftover block
            !            convertStatus := StrToVal(messageArray{posInStr},leftOverArray{i,1});
            !            posInStr := posInStr + 1;
            !            !y coordinate of leftover block
            !            convertStatus := StrToVal(messageArray{posInStr},leftOverArray{i,2});
            !            posInStr := posInStr + 1;
            !            !z coordinate of leftover block
            !            convertStatus := StrToVal(messageArray{posInStr},leftOverArray{i,3});
            !            posInStr := posInStr + 1;
            !            !x coordinate of junk area
            !            convertStatus := StrToVal(messageArray{posInStr},leftOverArray{i,4});
            !            posInStr := posInStr + 1;
            !            !y coordinate of junk area
            !            convertStatus := StrToVal(messageArray{posInStr},leftOverArray{i,5});
            !            posInStr := posInStr + 1;
            !            !z coordinate of junk area
            !            convertStatus := StrToVal(messageArray{posInStr},leftOverArray{i,6});
            !            posInStr := posInStr + 1;
            !            count := count + 1;
        ENDFOR

    ENDPROC

    ! INPUT
    !   string message - message which is to be SplitStr
    ! OUTPUT
    !   string messageArray{*} - Array of strings which contain the message
    ! NOTES
    !   Due to changes in how messages are sent, SplitStr is unused and replaced by receiveMessage
    PROC SplitStr(VAR string message,VAR string messageArray{*})
        VAR string delimiter:=",";
        VAR string buffer:="";
        VAR string char:="";
        VAR num len;

        VAR num charCount:=1;
        VAR num numStrings:=1;

        len:=StrLen(message);
        WHILE (charCount<=len) DO
            char:=StrPart(message,1,charCount);


            IF (char=",") THEN

                messageArray{numStrings}:=buffer;
                buffer:="";
                numStrings:=numStrings+1;
            ELSE
                buffer:=buffer+Char;
            ENDIF

            charCount:=charCount+1;
        ENDWHILE


    ENDPROC

! light curtain trap routine
    TRAP lTrap
        ! stop the robot & conveyor
        StopMove;
        IF DOutput(DO10_3)=1 THEN
            turnOffConveyor;
            tempConv:=1;
        ENDIF
        ! print message to gui
        lightCurtainError:=TRUE;
        ! print message to flex pendant
        TPErase;
        TPWrite "Light curtain obstruction";
        TPReadFK response,"Please remove obstruction",stEmpty,stEmpty,stEmpty,"No","Fixed";
        IF response=4 THEN
            TPErase;
            TPWrite "Exiting program...";
            WaitTime 2;
            EXIT;
        ELSEIF response=5 THEN
            TPErase;
            TPWrite "Resuming...";
            clearMessage:=TRUE;
        ENDIF
        StartMove;
        IF tempConv=1 THEN
            turnOnConveyor;
            tempConv:=0;
        ENDIF
        lightCurtainError:=FALSE;
        RETURN ;
    ENDTRAP

    ! emergency stop interrupt for red buttons except motor
    TRAP eTrap
        ! stop the robot
        StopMove;
        IF DOutput(DO10_3)=1 THEN
            turnOffConveyor;
            tempConv:=1;
        ENDIF
        ! print message to gui
        emergencyStopError:=TRUE;
        ! print message to flex pendant
        TPErase;
        TPWrite "Emergency stop!";
        TPWrite "Please remove any obstructions and hazards from the robot.";
        TPWrite "Don't forget to reset the light curtain.";
        TPReadFK response,"Restart?",stEmpty,stEmpty,stEmpty,"No","Yes";
        IF response=4 THEN
            TPErase;
            TPWrite "Exiting program...";
            WaitTime 2;
            EXIT;
        ELSEIF response=5 THEN
            TPErase;
            TPWrite "Resuming...";
            clearMessage:=TRUE;
        ENDIF
        StartMove;
        IF tempConv=1 THEN
            turnOnConveyor;
            tempConv:=0;
        ENDIF
        emergencyStopError:=FALSE;
        RETURN ;
    ENDTRAP

    ! emergency stop interrupt for motor button
    TRAP eTrapMotor
        ! stop the robot
        StopMove;
        IF DOutput(DO10_3)=1 THEN
            turnOffConveyor;
            tempConv:=1;
        ENDIF
        ! print message to gui
        emergencyStopError:=TRUE;
        ! print message to flex pendant
        TPErase;
        TPWrite "Motor stop!";
        TPWrite "Please remove any obstructions and hazards from the robot.";
        TPWrite "Don't forget to reset the light curtain.";
        TPReadFK response,"Restart?",stEmpty,stEmpty,stEmpty,"No","Yes";
        IF response=4 THEN
            TPErase;
            TPWrite "Exiting program...";
            WaitTime 2;
            EXIT;
        ELSEIF response=5 THEN
            TPErase;
            TPWrite "Resuming...";
            clearMessage:=TRUE;
        ENDIF
        StartMove;
        IF tempConv=1 THEN
            turnOnConveyor;
            tempConv:=0;
        ENDIF
        emergencyStopError:=FALSE;
        RETURN ;
    ENDTRAP

ENDMODULE

--- Backups/Vinnie/RAPID/TASK2/SYSMOD/MTRN_Rob_Data.sys ---
MODULE MTRN_Rob_Data (SYSMODULE, NOSTEPIN, READONLY)

 ! PREDEFINED DATA AND ROBOT CELL INFORMATION
 !*******************************************

 ! For the ABB IRB120 Robot in the Mechatronics Blockhouse Lab for the MTRN4230 Robotics Course 2014

 ! TARGETS
 !********

 ! Calibrate Position for all Joints
 CONST jointtarget jtCalibPos:=[[-90,0,0,0,0,0],[9E+09,9E+09,9E+09,9E+09,9E+09,9E+09]];

 ! Home Position of the Table (T1) with tSCup touching Table
 CONST robtarget pTableHome:=[[175,0,147],[0,0,-1,0],[0,0,0,0],[9E+09,9E+09,9E+09,9E+09,9E+09,9E+09]];

 ! Home Position of the Conveyor (C1) with tSCup touching Conveyor
 CONST robtarget pConvHome:=[[0,409,22],[0,-0.7071068,0.7071068,0],[0,0,0,0],[9E+09,9E+09,9E+09,9E+09,9E+09,9E+09]];

 ! Table & Conveyor Dimensions, References & Extent limits as Follows (X,Y,Z in mm):
 !
 !                                                       Conveyor Frame
 !       ------>Y                                   |<-------- 616 -------->|
 !       |                                          |   | Conveyor Belt |   |
 !       |                                          |   |<---- 450 ---->|   |
 !       |                            ||    --------|   |               |   |
 !       v                            \/    |------||   |   0,409,22    |   |
 !       X             Robot Centre  ---->  ||  + |||   |      +        |   |
 !                                          ||    |||   |      C1       |   |
 !     Robot Centre to edge of Table=129    -|    |_|   |               |   |
 !   ----------------------------------------|    |-----------------------------------
 !   |                                /\      ----                                   |
 !   |                                ||      |  |                                   |
 !   |     175,-520,147                     175,0,147                  175,520,147   |
 !   |           +                              +                           +        |
 !   |           T2                             T1                          T3       |
 !   |                                                                               |
 !   |                                                                               |
 !   |                                    548.6,0,147                                |
 !   |                                          +                                    |
 !   |                                          T4                                   |
 !   |                                                                               |
 !   ---------------------------------------------------------------------------------

 ! TOOL DATA
 !**********

 ! Suction Cup Tool Data
 PERS tooldata tSCup:=[TRUE,[[0,0,65],[1,0,0,0]],[0.5,[0,0,20],[1,0,0,0],0,0,0]];
 !
 ! Suction Cup Face is 65mm in Z direction from Tool0

 ! LOAD DATA
 !**********

 ! Chocolate Bar Load Data
 PERS loaddata loChoc:=[0.035,[0,0,3],[1,0,0,0],0,0,0];

 !
 ! Chocolate Bar Weight    : 35g
 !
 ! Chocolate Bar Dimensions: 114.5 x 53 x 7.5mm (Including Perspex substitute in wrapper)
 !
 ! Chocolate Box Dimensions: 214.0 x 119.0 x 46.0mm (Internal)
 !                           219.5 x 121.0 x 48.0mm (External)
 !
 ! Chocolate Box References:
 !
 !                         -------------------------
 !                         |----- ----- ----- -----|
 !                         ||   | |   | |   | |   ||
 !                         ||   | |   | |   | |   ||
 !                         ||B4 | |B3 |+|B2 | |B1 ||
 !                         ||   | |   | |   | |   ||
 !                         ||   | |   | |   | |   ||
 !                         |----- ----- ----- -----|
 !                         -------------------------
 !
 ! NOTE: + marks centre of box and Conveyor Home Position C1

 ! WORK OBJECT DATA
 !*****************
 !                                    [Uframe User co-ord System] [Oframe Object Co-ord System]
 PERS wobjdata wTable:=[FALSE,TRUE,"",[[175,0,147],[1,0,0,0]],[[0,0,0],[1,0,0,0]]];
 PERS wobjdata wConv:=[FALSE,TRUE,"",[[50,184,22],[0.5,-0.5,0.5,0.5]],[[1,1,1],[1,0,0,0]]];

 ! WorkObject orientations for the Table and Conveyor
 !
 !                    |   |               |   |
 !                    |   Y               |   |
 !                    |   ^               |   |
 !             -------|   |               |   |
 !             |     ||   | \Wobj:=vConv  |   |
 !             |  +  ||   |               |   |
 !             |     ||   |               |   |
 !             -------|  Zo------>X       |   |
 !   ---------------------------------------------------
 !               Zo----->Y                             |
 !                |                                    |
 !                | \Wobj:=vTable                      |
 !                |                                    |
 !                v                                    |
 !                X                                    |
 !                                                     |

 ! COMMENTS
 !*********

 ! Digital I/O Names and Functions
 ! DI10-1	ConStat	= Conveyor Status (Active = 1, Inactive = 0)
 !
 ! DO10-1	VacPwr	= Vacuum Power (Run = 1, Stop =0)
 ! DO10-2	VacSol	= Vacuum Solenoid (Open = 1, Closed =0)
 ! D010-3	ConRun	= Conveyer Start (Run = 1, Stop = 0)
 ! D010-4	ConDir	= Conveyer Direction (Towards Robot = 1, Away from Robot = 0)

ENDMODULE

--- Backups/Vinnie/RAPID/TASK2/SYSMOD/MTRN_Rob_Proc.sys ---
MODULE MTRN_Rob_Proc (SYSMODULE, NOSTEPIN, READONLY)

 ! MTRN ROBOTICS COMMON PROCEDURES
 !********************************
 !
 ! For the ABB IRB120 Robot in the Mechatronics Blockhouse Lab for the MTRN4230 Robotics Course 2014
 !

 PROC MoveToCalibPos()
 !***************************************************************************************
 !
 ! Move to Calibrate Position
 !
 !***************************************************************************************

 MoveAbsJ jtCalibPos,v400,fine,tool0;

 ENDPROC

ENDMODULE

--- Backups/Vinnie/HOME/MTRN4230_Move_Sample.mod ---
MODULE MTRN4230_Move_Sample

    ! The Main procedure. When you select 'PP to Main' on the FlexPendant, it will go to this procedure.
    PROC MainMove()

        ! This is a procedure defined in a System Module, so you will have access to it.
        ! This will move the robot to its calibration.
        MoveToCalibPos;

        ! Call a procedure that we have defined below.
        MoveJSample;

        ! Call another procedure that we have defined.
        MoveLSample;

        ! Call another procedure, but provide some input arguments.
        VariableSample pTableHome, 100, 100, 0, v100, fine;

    ENDPROC

    PROC MoveJSample()

        ! 'MoveJ' executes a joint motion towards a robtarget. This is used to move the robot quickly from one point to another when that
        !   movement does not need to be in a straight line.
        ! 'pTableHome' is a robtarget defined in system module. The exact location of this on the table has been provided to you.
        ! 'v100' is a speeddata variable, and defines how fast the robot should move. The numbers is the speed in mm/sec, in this case 100mm/sec.
        ! 'fine' is a zonedata variable, and defines how close the robot should move to a point before executing its next command.
        !   'fine' means very close, other values such as 'z10' or 'z50', will move within 10mm and 50mm respectively before executing the next command.
        ! 'tSCup' is a tooldata variable. This has been defined in a system module, and represents the tip of the suction cup, telling the robot that we
        !   want to move this point to the specified robtarget. Please be careful about what tool you use, as using the incorrect tool will result in
        !   the robot not moving where you would expect it to. Generally you should be using
        MoveJ pTableHome, v100, fine, tSCup;

    ENDPROC

    PROC MoveLSample()

        ! 'MoveL' will move in a straight line between 2 points. This should be used as you approach to pick up a chocolate
        ! 'Offs' is a function that is used to offset an existing robtarget by a specified x, y, and z. Here it will be offset 100mm in the positive z direction.
        !   Note that function are called using brackets, whilst procedures and called without brackets.
        MoveL Offs(pTableHome, 0, 0, 0), v100, fine, tSCup;

    ENDPROC

    PROC VariableSample(robtarget target, num x_offset, num y_offset, num z_offset, speeddata speed, zonedata zone)

        ! Call 'MoveL' with the input arguments provided.
        MoveL Offs(target, x_offset, y_offset, z_offset), speed, zone, tSCup;

    ENDPROC

ENDMODULE

--- Backups/Vinnie/HOME/MTRN4230_Server_Sample.mod ---
MODULE MTRN4230_Server_Sample

    ! The socket connected to the client.
    VAR socketdev client_socket;

    ! The host and port that we will be listening for a connection on.
    PERS string host := "192.168.125.1";

    CONST num port := 1025;

    PROC Main ()
        IF RobOS() THEN
            host := "192.168.125.1";
        ELSE
            host := "127.0.0.1";
        ENDIF
        MainServer;

    ENDPROC

    PROC MainServer()

        VAR string received_str;

        ListenForAndAcceptConnection;

        ! Receive a string from the client.
        SocketReceive client_socket \Str:=received_str;

        ! Send the string back to the client, adding a line feed character.
        SocketSend client_socket \Str:=(received_str + "\0A");

        CloseConnection;

    ENDPROC

    PROC ListenForAndAcceptConnection()

        ! Create the socket to listen for a connection on.
        VAR socketdev welcome_socket;
        SocketCreate welcome_socket;

        ! Bind the socket to the host and port.
        SocketBind welcome_socket, host, port;

        ! Listen on the welcome socket.
        SocketListen welcome_socket;

        ! Accept a connection on the host and port.
        SocketAccept welcome_socket, client_socket \Time:=WAIT_MAX;

        ! Close the welcome socket, as it is no longer needed.
        SocketClose welcome_socket;

    ENDPROC

    ! Close the connection to the client.
    PROC CloseConnection()
        SocketClose client_socket;
    ENDPROC


ENDMODULE

--- Backups/Vinnie/SYSPAR/EIO.cfg ---
EIO:CFG_1.0:5:0::
#
EIO_BUS:

      -Name "Virtual1" -ConnectorID "SIM1"

      -Name "DeviceNet_Lean" -BusType "DNLE" -ConnectorID "PCI1"\
      -ConnectorLabel "DeviceNet Lean"
#
EIO_UNIT_TYPE:

      -Name "Virtual" -VendorName "ABB" -ProductName "Virtual unit"

      -Name "d651_Lean" -BusType "DNLE" -VendorName "ABB Robotics"\
      -ProductName "Combi Unit" -DL_ProductCode 25

      -Name "d652_Lean" -BusType "DNLE" -VendorName "ABB Robotics"\
      -ProductName "24 VDC Unit" -DL_ProductCode 26

      -Name "d653_Lean" -BusType "DNLE" -VendorName "ABB Robotics"\
      -ProductName "Relay Unit" -DL_ProductCode 27

      -Name "AC500_PLC_Lean" -BusType "DNLE" -VendorName "ABB Stotz"\
      -ProductName "AC500 PLC - FPB" -DL_ProductCode 1 -DL_VendorID 760

      -Name "DL_GENERIC" -BusType "DNLE" -DL_ProductCode 3535

      -Name "DL_GENERIC_POLL" -BusType "DNLE" -DL_ProductCode 3535\
      -DL_Pollrate 30

      -Name "d351_Lean" -BusType "DNLE" -VendorName "ABB Robotics"\
      -ProductName "IBS Adapter" -DL_ProductCode 7

      -Name "d352_Lean" -BusType "DNLE" -VendorName "ABB Robotics"\
      -ProductName "PBUS Adapter" -DL_ProductCode 8

      -Name "d378_Lean" -BusType "DNLE" -VendorName "ABB Robotics"\
      -ProductName "CCLink Adapter" -DL_ProductCode 17
#
EIO_UNIT:

      -Name "BOARD10" -UnitType "d652_Lean" -Bus "DeviceNet_Lean" -DL_Address 10
#
EIO_SIGNAL:

      -Name "DI10_1" -SignalType "DI" -Unit "BOARD10" -SignalLabel "ConStat"\
      -UnitMap "0"

      -Name "DI10_2" -SignalType "DI" -Unit "BOARD10" -UnitMap "1"

      -Name "DI10_3" -SignalType "DI" -Unit "BOARD10" -UnitMap "2"

      -Name "DI10_4" -SignalType "DI" -Unit "BOARD10" -UnitMap "3"

      -Name "DI10_5" -SignalType "DI" -Unit "BOARD10" -UnitMap "4"

      -Name "DI10_6" -SignalType "DI" -Unit "BOARD10" -UnitMap "5"

      -Name "DI10_7" -SignalType "DI" -Unit "BOARD10" -UnitMap "6"

      -Name "DI10_8" -SignalType "DI" -Unit "BOARD10" -UnitMap "7"

      -Name "DI10_9" -SignalType "DI" -Unit "BOARD10" -UnitMap "8"

      -Name "DI10_10" -SignalType "DI" -Unit "BOARD10" -UnitMap "9"

      -Name "DI10_11" -SignalType "DI" -Unit "BOARD10" -UnitMap "10"

      -Name "DI10_12" -SignalType "DI" -Unit "BOARD10" -UnitMap "11"

      -Name "DI10_13" -SignalType "DI" -Unit "BOARD10" -UnitMap "12"

      -Name "DI10_14" -SignalType "DI" -Unit "BOARD10" -UnitMap "13"

      -Name "DI10_15" -SignalType "DI" -Unit "BOARD10" -UnitMap "14"

      -Name "DI10_16" -SignalType "DI" -Unit "BOARD10" -UnitMap "15"\
      -Access "All"

      -Name "DO10_1" -SignalType "DO" -Unit "BOARD10" -SignalLabel "VacRun"\
      -UnitMap "0"

      -Name "DO10_2" -SignalType "DO" -Unit "BOARD10" -SignalLabel "VacSol"\
      -UnitMap "1"

      -Name "DO10_3" -SignalType "DO" -Unit "BOARD10" -SignalLabel "ConRun"\
      -UnitMap "2"

      -Name "DO10_4" -SignalType "DO" -Unit "BOARD10" -SignalLabel "ConDir"\
      -UnitMap "3"

      -Name "DO10_5" -SignalType "DO" -Unit "BOARD10" -UnitMap "4"

      -Name "DO10_6" -SignalType "DO" -Unit "BOARD10" -UnitMap "5"

      -Name "DO10_7" -SignalType "DO" -Unit "BOARD10" -UnitMap "6"

      -Name "DO10_8" -SignalType "DO" -Unit "BOARD10" -UnitMap "7"

      -Name "DO10_9" -SignalType "DO" -Unit "BOARD10" -UnitMap "8"

      -Name "DO10_10" -SignalType "DO" -Unit "BOARD10" -UnitMap "9"

      -Name "DO10_11" -SignalType "DO" -Unit "BOARD10" -UnitMap "10"

      -Name "DO10_12" -SignalType "DO" -Unit "BOARD10" -UnitMap "11"

      -Name "DO10_13" -SignalType "DO" -Unit "BOARD10" -UnitMap "12"

      -Name "DO10_14" -SignalType "DO" -Unit "BOARD10" -UnitMap "13"

      -Name "DO10_15" -SignalType "DO" -Unit "BOARD10" -UnitMap "14"

      -Name "DO10_16" -SignalType "DO" -Unit "BOARD10" -UnitMap "15"

      -Name "DO_LIGHT_CURTAIN" -SignalType "DO" -Access "ReadOnly"

      -Name "DO_ESTOP" -SignalType "DO" -Access "ReadOnly"

      -Name "DO_MOTION_SUP_TRIG" -SignalType "DO" -Access "ReadOnly"

      -Name "DO_MOTOR_ON_STATE" -SignalType "DO" -Access "ReadOnly"

      -Name "DO_EXEC_ERR" -SignalType "DO" -Access "ReadOnly"

      -Name "DO_TROB_RUNNING" -SignalType "DO" -Access "ReadOnly"

      -Name "DO_HOLD_TO_ENABLE" -SignalType "DO" -Access "ReadOnly"

      -Name "DI_MOTOR_ON" -SignalType "DI" -Access "ReadOnly"

      -Name "DO_ESTOP2" -SignalType "DO" -Access "ReadOnly"
#
EIO_CROSS:

      -Res "DO_LIGHT_CURTAIN" -Act1 "GS1" -Oper1 "AND" -Act2 "GS2"

      -Res "DO_HOLD_TO_ENABLE" -Act1 "EN1" -Oper1 "AND" -Act2 "EN2"

      -Res "DI_MOTOR_ON" -Act1 "MONPB"

      -Res "DO_ESTOP" -Act1 "ES1" -Oper1 "AND" -Act2 "ES2"
#
EIO_COMMAND_TYPE:

      -Name "DataWidth_L" -UnitType "d351_Lean" -DefValue "3" -OrderNr 1\
      -DL_Path "6,20 65 24 01 30 01,C6,1"

      -Name "D351reset_L" -UnitType "d351_Lean" -DefValue "0" -OrderNr 2\
      -DL_Path "4,20 01 24 01,C1,1" -DL_Service 5

      -Name "MasterInputSize_B_L" -UnitType "d352_Lean" -DefValue "1" -OrderNr 1\
      -DL_Path "6,20 67 24 01 30 02,C6,1"

      -Name "MasterOutputSize_B_L" -UnitType "d352_Lean" -DefValue "1"\
      -OrderNr 2 -DL_Path "6,20 67 24 01 30 03,C6,1"

      -Name "StationAddress_B_L" -UnitType "d352_Lean" -DefValue "126"\
      -OrderNr 3 -DL_Path "6,20 67 24 01 30 04,C6,1"

      -Name "D352reset_L" -UnitType "d352_Lean" -DefValue "0" -OrderNr 4\
      -DL_Path "4,20 01 24 01,C1,1" -DL_Service 5

      -Name "StationNo_L" -UnitType "d378_Lean" -DefValue "1" -OrderNr 1\
      -DL_Path "6,20 68 24 01 30 01,C6,1"

      -Name "BaudRate_L" -UnitType "d378_Lean" -DefValue "0" -OrderNr 2\
      -DL_Path "6,20 68 24 01 30 02,C6,1"

      -Name "OccStat_L" -UnitType "d378_Lean" -DefValue "1" -OrderNr 3\
      -DL_Path "6,20 68 24 01 30 03,C6,1"

      -Name "BasicIO_L" -UnitType "d378_Lean" -DefValue "0" -OrderNr 4\
      -DL_Path "6,20 68 24 01 30 04,C1,1"

      -Name "D378reset_L" -UnitType "d378_Lean" -DefValue "0" -OrderNr 5\
      -DL_Path "4,20 01 24 01,C1,1" -DL_Service 5
#
EIO_ACCESS:

      -Name "All" -Rapid  -LocalManual  -LocalAuto  -RemoteManual  -RemoteAuto
#
SYSSIG_OUT:

      -Status "EmStop" -Signal "DO_ESTOP2"

      -Status "MotSupTrigg" -Signal "DO_MOTION_SUP_TRIG" -Arg1 "ROB_1"

      -Status "MotOnState" -Signal "DO_MOTOR_ON_STATE"

      -Status "Error" -Signal "DO_EXEC_ERR" -Arg2 "T_ROB1"

      -Status "TaskExecuting" -Signal "DO_TROB_RUNNING" -Arg2 "T_ROB1"

--- Backups/Vinnie/SYSPAR/PROC.cfg ---
PROC:CFG_1.0:5:0::
#
GAP_TASK_NAME_MAPPING:

      -name "T_ROB1" -common_name "T_ROB1" -tab_index 1
